(* CODESYS project Johnson,Joachim,Uppgift17_V1.project

Project tree, tasks and I/O mapping:
  Device : CODESYS Control Win V3, 3S - Smart Software Solutions GmbH, order no. 305021, version 3.5.10.40
    application Application
      libraries: Standard, * (System)
      task MainTask (cyclic, interval t#20ms, priority 1) calls PLC_PRG
      program PLC_PRG [SFC]: MoveConv1to2, MoveCon2to3, Setrunning, SetStop, StopBTNCHECK, ResetAlarm
      global variables GVL
      Symbols
*)

// Device/Application/GVL
{attribute 'qualified_only'}
VAR_GLOBAL
	// signals from buttons
	iSUB00_S1: BOOL; // StartButton
	iSUB00_S2: BOOL; // Stopbutton
	iSUB00_S3: BOOL; // Resetbutton
	
	running: BOOL; // Is the aplication running
	alarm: BOOL; // Is the aplication running
	
	// Signals from conveyors
	iSUB01_B1: BOOL; // Signals för conveyor 1. ontop
	iSUB02_B1: BOOL; // Signals för conveyor 2. ontop
	iSUB03_B1: BOOL; // Signals för conveyor 3. ontop
	
	// conveyor signal ontop conveyro.
	oSUB00_H1: BOOL; // Auto-On light
	oSUB00_H2: BOOL; // Alarm light
	oSUB00_H3: BOOL;
	oSUB01_K1: BOOL; // MOTOR FÖR converoyr 1
	oSUB02_K1: BOOL; // MOTOR FÖR converoyr 2
	oSUB03_K1: BOOL; // MOTOR FÖR converoyr 3
END_VAR

// Device/Application/PLC_PRG
PROGRAM PLC_PRG
VAR	
	TON_0: TON;
	OutputTime: TIME;
	TON2: TON;
	Output: TIME;
END_VAR
VAR // added by the converter: edge detectors and wires of the graphical bodies
    _w1, _w3, _w5, _w6 : BOOL;
    _w2, _w4, _w7, _w8, _w9, _w10 : ANY;
END_VAR

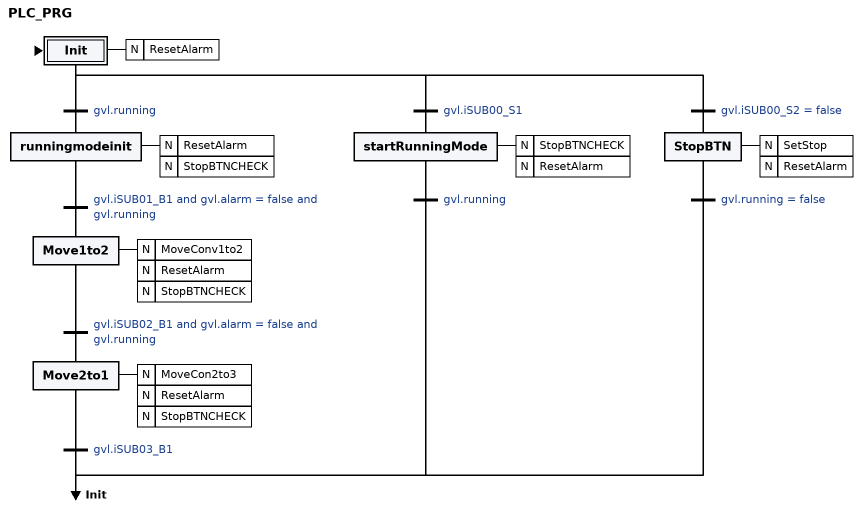
INITIAL_STEP Init:
    ResetAlarm(N);
END_STEP
TRANSITION FROM Init TO runningmodeinit
    := gvl.running;
END_TRANSITION
STEP runningmodeinit:
    ResetAlarm(N);
    StopBTNCHECK(N);
END_STEP
TRANSITION FROM runningmodeinit TO Move1to2
    := gvl.iSUB01_B1 and gvl.alarm = false and gvl.running;
END_TRANSITION
STEP Move1to2:
    MoveConv1to2(N);
    ResetAlarm(N);
    StopBTNCHECK(N);
END_STEP
TRANSITION FROM Move1to2 TO Move2to1
    := gvl.iSUB02_B1 and gvl.alarm = false and gvl.running;
END_TRANSITION
STEP Move2to1:
    MoveCon2to3(N);
    ResetAlarm(N);
    StopBTNCHECK(N);
END_STEP
TRANSITION FROM Move2to1 TO Init
    := gvl.iSUB03_B1;
END_TRANSITION
TRANSITION FROM Init TO startRunningMode
    := gvl.iSUB00_S1;
END_TRANSITION
STEP startRunningMode:
    StopBTNCHECK(N);
    ResetAlarm(N);
END_STEP
TRANSITION FROM startRunningMode TO Init
    := gvl.running;
END_TRANSITION
TRANSITION FROM Init TO StopBTN
    := gvl.iSUB00_S2 = false;
END_TRANSITION
STEP StopBTN:
    SetStop(N);
    ResetAlarm(N);
END_STEP
TRANSITION FROM StopBTN TO Init
    := gvl.running = false;
END_TRANSITION

ACTION MoveConv1to2:
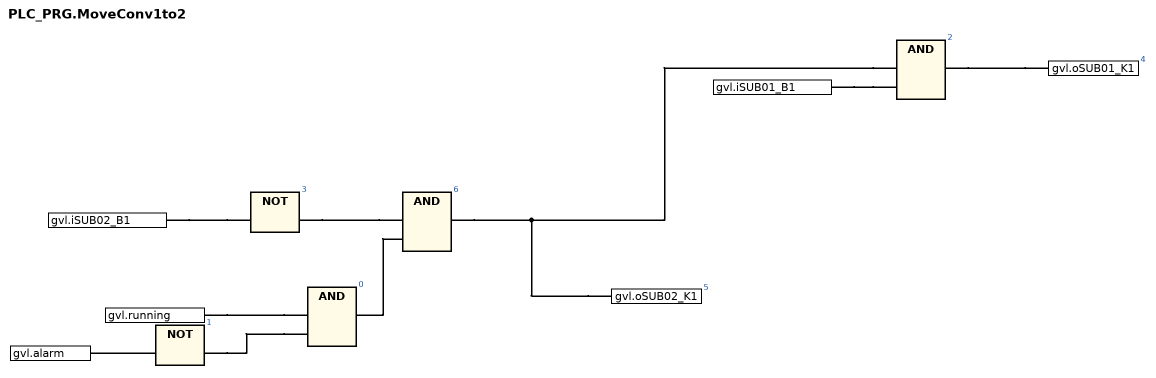
_w2 := gvl.running AND _w1;
_w1 := NOT gvl.alarm;
_w4 := NOT gvl.iSUB02_B1;
gvl.oSUB01_K1 := _w3 AND gvl.iSUB01_B1;
gvl.oSUB02_K1 := _w3;
_w3 := _w4 AND _w2;
END_ACTION

ACTION MoveCon2to3:
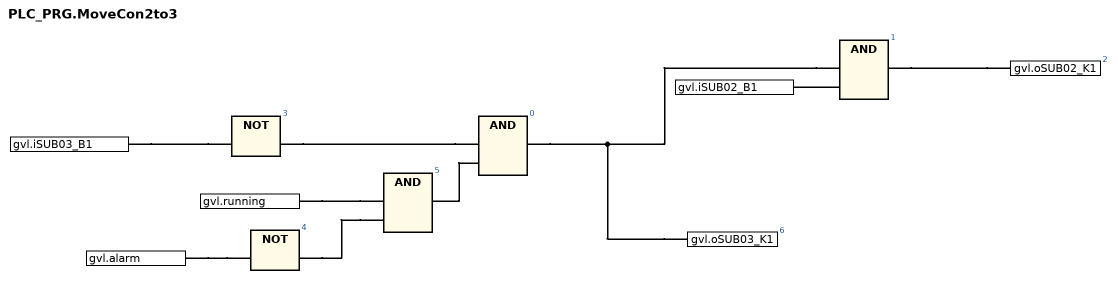
_w7 := _w5 AND _w6;
gvl.oSUB02_K1 := _w7 AND gvl.iSUB02_B1;
_w5 := NOT gvl.iSUB03_B1;
_w6 := gvl.running AND NOT gvl.alarm;
gvl.oSUB03_K1 := _w7;
END_ACTION

ACTION Setrunning:
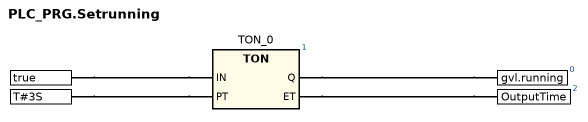
gvl.running := TON_0.Q;
TON_0(IN := true, PT := T#3S); // TON
OutputTime := TON_0.ET;
END_ACTION

ACTION SetStop:
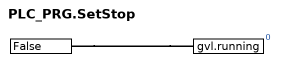
gvl.running := False;
END_ACTION

ACTION StopBTNCHECK:
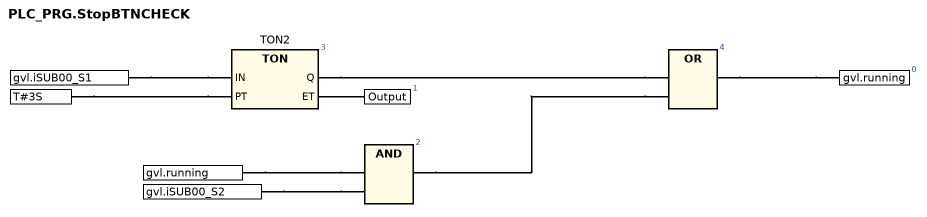
gvl.running := _w8;
Output := TON2.ET;
_w9 := gvl.running AND gvl.iSUB00_S2;
TON2(IN := gvl.iSUB00_S1, PT := T#3S); // TON
_w8 := TON2.Q OR _w9;
END_ACTION

ACTION ResetAlarm:
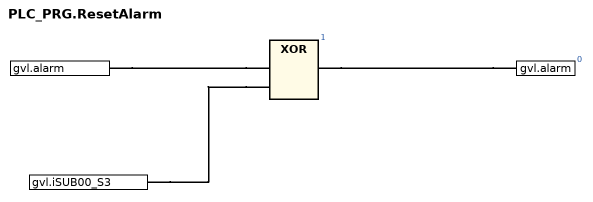
gvl.alarm := _w10;
_w10 := gvl.alarm XOR gvl.iSUB00_S3;
END_ACTION

END_PROGRAM
